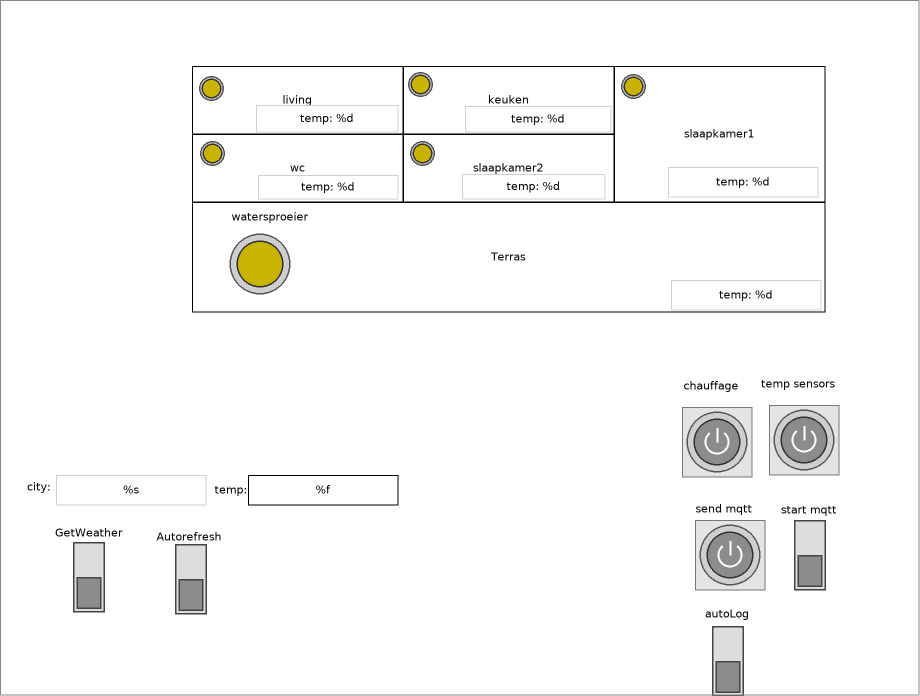
VISUALIZATION Visualization  // 920x696
    Rectangle (192,66 211x68), "living", colour toggle: MAIN.living.Lamp1
        tap MAIN.living.schakelaar
    Rectangle (403,66 211x68), "keuken", colour toggle: MAIN.keuken.Lamp1
        tap MAIN.keuken.schakelaar
    Rectangle (192,134 211x68), "wc", colour toggle: MAIN.wc.Lamp1
        tap MAIN.wc.schakelaar
    Rectangle (403,134 211x68), "slaapkamer2", colour toggle: MAIN.slaapkamer2.Lamp1
        tap MAIN.slaapkamer2.schakelaar
    Rectangle (614,66 211x136), "slaapkamer1", colour toggle: MAIN.slaapkamer1.Lamp1
        tap MAIN.slaapkamer1.schakelaar
    Textfield (668,167 150x30), "temp: %d", text variable: MAIN.slaapkamer1.tempValue, invisible if: not MAIN.temp
        OnMouseDown: write the text variable via Default
    Textfield (462,174 143x25), "temp: %d", text variable: MAIN.slaapkamer2.tempValue, invisible if: not MAIN.temp
        OnMouseDown: write the text variable via Default
    Textfield (465,106 146x26), "temp: %d", text variable: MAIN.keuken.tempValue, invisible if: not MAIN.temp
        OnMouseDown: write the text variable via Default
    Textfield (256,105 142x27), "temp: %d", text variable: MAIN.living.tempValue, invisible if: not MAIN.temp
        OnMouseDown: write the text variable via Default
    Textfield (258,175 140x24), "temp: %d", text variable: MAIN.wc.tempValue, invisible if: not MAIN.temp
        OnMouseDown: write the text variable via Default
    PowerSwitch (769,405 70x70), variable: MAIN.temp, behaviour: TOGGLE, style: Switch-PowerSwitch-Gray
    Rectangle (192,202 633x110), "Terras", colour toggle: MAIN.terras.Lamp1
        tap MAIN.terras.schakelaar
    Textfield (671,280 150x30), "temp: %d", text variable: MAIN.terras.tempValue, invisible if: not MAIN.temp
        OnMouseDown: write the text variable via Default
    Lamp1 (196,74 31x29), variable: MAIN.living.chauffage, style: Lamp-Lamp1-Yellow
    Lamp1 (197,139 31x29), variable: MAIN.wc.chauffage, style: Lamp-Lamp1-Yellow
    Lamp1 (405,70 31x29), variable: MAIN.keuken.chauffage, style: Lamp-Lamp1-Yellow
    Lamp1 (618,72 31x29), variable: MAIN.slaapkamer1.chauffage, style: Lamp-Lamp1-Yellow
    Lamp1 (407,139 31x29), variable: MAIN.slaapkamer2.chauffage, style: Lamp-Lamp1-Yellow
    Label (723,369 150x30), "temp sensors"
    PowerSwitch (682,407 70x70), variable: MAIN.chauffageOn, behaviour: TOGGLE, style: Switch-PowerSwitch-Gray
    DipSwitch (54,542 70x70), variable: MAIN.bGetOpenWeatherMap, behaviour: TOGGLE, style: Switch-DipSwitch-Gray
    Textfield (56,475 150x30), "%s", text variable: MAIN.GetValues.city
        OnMouseClick: write the text variable via Default
    Rectangle (248,475 150x30), "%f", text variable: MAIN.GetValues.sTemp
    Label (210,478 42x24), "temp:"
    Label (-36,472 150x30), "city:"
    DipSwitch (775,520 70x70), variable: MQTT.startbutton, behaviour: TOGGLE, style: Switch-DipSwitch-Gray
    PowerSwitch (695,520 70x70), variable: MQTT.sendbutton, behaviour: TAP, style: Switch-PowerSwitch-Gray
    Label (734,495 150x30), "start mqtt"
    Label (649,494 150x30), "send mqtt"
    Lamp1 (225,229 70x70), variable: main.terras.watersproeier, style: Lamp-Lamp1-Yellow
    Label (195,202 150x30), "watersproeier"
    DipSwitch (693,626 70x70), tooltip "autoLog", variable: MAIN.logs, behaviour: TOGGLE, style: Switch-DipSwitch-Gray
    Label (652,599 150x30), "autoLog"
    DipSwitch (156,544 70x70), tooltip "autorefresh", variable: autorefresh, behaviour: TOGGLE, style: Switch-DipSwitch-Gray
    Label (14,518 150x30), "GetWeather"
    Label (114,522 150x30), "Autorefresh"
    Label (636,371 150x30), "chauffage"
END_VISUALIZATION

(* stored: Version 1.1.0.1, ProductVersion 3.1.4024.9
   Visu Visualization: Id {0da14ef1-a9d4-46c2-b271-b5c61610efc9} *)
